(* CODESYS project outputs.project

Project tree, tasks and I/O mapping:
  Device : CODESYS Control Win V3 x64, 3S - Smart Software Solutions GmbH, version 3.5.11.0
    application Application
      libraries: Standard, * (System); VisuDialogs, * (System); Util, * (System)
      task MainTask (cyclic, interval t#10ms, priority 1) calls Plant, Controller
      program Plant [ST]
      global variables GVL
      program Controller [ST]
      visualisation Visualization
      image pool ImagePool
  text list GlobalTextList
  5ce3da45-db07-42e7-a21c-a00fff4ed8f6|C:\Users\mihas\Documents\NSU2026\AM\images\input\beer.png
  5ce3da45-db07-42e7-a21c-a00fff4ed8f6|C:\Users\mihas\Documents\NSU2026\AM\images\input\cigaretes after vki .png
  5ce3da45-db07-42e7-a21c-a00fff4ed8f6|C:\Users\mihas\Documents\NSU2026\AM\images\input\greencard.png
  5ce3da45-db07-42e7-a21c-a00fff4ed8f6|C:\Users\mihas\Documents\NSU2026\AM\images\input\jaguar.png
  5ce3da45-db07-42e7-a21c-a00fff4ed8f6|C:\Users\mihas\Documents\NSU2026\AM\images\input\monster.png
  5ce3da45-db07-42e7-a21c-a00fff4ed8f6|C:\Users\mihas\Documents\NSU2026\AM\images\input\pistol.png
  5ce3da45-db07-42e7-a21c-a00fff4ed8f6|C:\Users\mihas\Documents\NSU2026\AM\images\input\voenbilet.png
*)

// Device/Application/GVL
VAR_GLOBAL
	// Sensors:
	onfloor0:BOOL;		// Elevator at floor 0
	onfloor1:BOOL;		// Elevator at floor 1
	onfloor2:BOOL;		// Elevator at floor 2
	door0closed:BOOL;	// Doors at floor 0 are closed
	door1closed:BOOL;	// Doors at floor 1 are closed
	door2closed:BOOL;	// Doors at floor 2 are closed
	button0:BOOL;		// Call button at floor 0
	button1:BOOL;		// Call button at floor 1
	button2:BOOL;		// Call button at floor 2
	call0:BOOL;			// Request floor 0 from inside the cabin 
	call1:BOOL;			// Request floor 1 from inside the cabin
	call2:BOOL;			// Request floor 2 from inside the cabin
	
	// Actuators:
	up:BOOL;			// Control the elevator to go up
	down:BOOL;			// Control the elevator to go down
	open0:BOOL;			// Open the doors at floor 0
	open1:BOOL;			// Open the doors at floor 1
	open2:BOOL;			// Open the doors at floor 2
	
	call0_LED : BOOL;
	call1_LED : BOOL;
	call2_LED : BOOL;
	
	button0_LED : BOOL;
	button1_LED : BOOL;
	button2_LED : BOOL;
	
	floor0_LED : BOOL;
	floor1_LED : BOOL;
	floor2_LED : BOOL;
	
	cur : INT;
END_VAR

// Device/Application/Plant
PROGRAM Plant

VAR
	cur : BOOL;
	dx : DINT;
	start_time_ms : DINT := TIME_TO_DINT(TIME());
	start_time_text : DINT := TIME_TO_DINT(TIME());
	start_time_angle : DINT := TIME_TO_DINT(TIME());
	angle : DINT := 0;

	sets: STRING := 'TIP TERMINAL';

	i : DINT := 0;
	
	text_welcome_message : WSTRING(250) := "Приветствуем тебя в Пивном Аппарате!!!$nВыбери товар, брат)";
	text_out_of_stock : WSTRING(250) := "В аппарате кончился выбранный товар, брат.$nЗаходи завтра, брат.";
	text_in_stock : WSTRING(250) := "Брат, товар, который ты хочешь есть в наличии.$nЩа оплатить только надо будет, брат.";
	text_insert_payment : WSTRING(250) := "Плати бабки за товар, брат.";
	text_not_enough_money : WSTRING(250) := "Добрось монеток, брат.$nСредств недостаточно.";
	text_stuff_not_dropped : WSTRING(250) := "Пружина не сработала, брат, либо возникла другая проблема.$nПозвони в поддержку, брат. Там всегда ждут твоего звонка";
	text_mission_completed : WSTRING(250) := "Братишка, у тебя получилось.$nНаслаждайся тяжелым люксом, брат!!!";
	
	text_arr : ARRAY[0..6] OF WSTRING(250) := [text_welcome_message, text_out_of_stock, text_in_stock, text_insert_payment, text_not_enough_money, text_stuff_not_dropped, text_mission_completed];
	
	text_display : WSTRING(1024) := text_welcome_message;
	
	Springs : ARRAY [0..4] OF BOOL := [FALSE, FALSE, FALSE, FALSE, FALSE];

END_VAR

dx := (TIME_TO_DINT(TIME()) - start_time_ms) / 1000;
IF ((TIME_TO_DINT(TIME())) - start_time_text) MOD 2000 > 1000 THEN 
	start_time_text := TIME_TO_DINT(TIME());
	IF i = 6 THEN
		i := 0;
	ELSE
		i := i + 1;	
	END_IF
	
	
END_IF

// Поворот пружины

IF ((TIME_TO_DINT(TIME())) - start_time_angle) MOD 2000 > (1000 / 25) THEN 
	start_time_angle := TIME_TO_DINT(TIME());
	angle := (angle + 360 / 25) MOD 360;
END_IF


text_display := text_arr[i];

END_PROGRAM

// Device/Application/Controller
PROGRAM Controller

VAR CONSTANT
	_STOP : INT := 254;
	_ERROR : INT := 255;
END_VAR

VAR
	target : INT;
END_VAR

END_PROGRAM

// Device/Application/Visualization
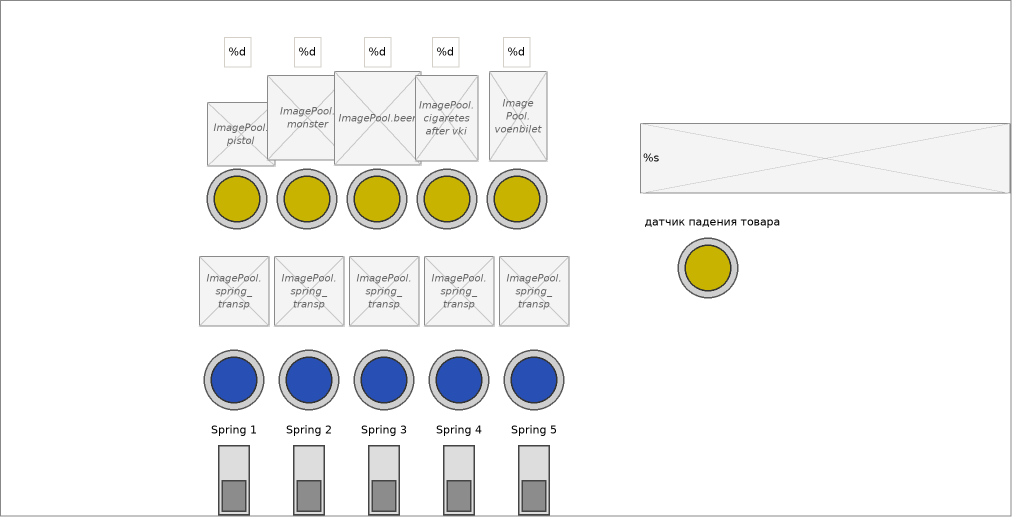
VISUALIZATION Visualization  // 1012x517
    Polygon (363,76) (364,77)
    Lamp1 (199,345 70x70), variable: Plant.Springs[0], style: Lamp-Lamp1-Blue
    Lamp1 (274,345 70x70), variable: Plant.Springs[1], style: Lamp-Lamp1-Blue
    Lamp1 (349,345 70x70), variable: Plant.Springs[2], style: Lamp-Lamp1-Blue
    Lamp1 (424,345 70x70), variable: Plant.Springs[3], style: Lamp-Lamp1-Blue
    Lamp1 (499,345 70x70), variable: Plant.Springs[4], style: Lamp-Lamp1-Blue
    DipSwitch (424,445 70x70), variable: Plant.Springs[3], behaviour: TOGGLE, style: Switch-DipSwitch-Gray
    Image (640,123 370x70), "%s", text variable: Plant.text_display, image: VisuDialogs.ImagePoolDialogs.Title
    Label (199,415 70x30), "Spring 1"
    Label (499,415 70x30), "Spring 5"
    Label (274,415 70x30), "Spring 2"
    Label (349,415 70x30), "Spring 3"
    Label (424,415 70x30), "Spring 4"
    DipSwitch (499,445 70x70), variable: Plant.Springs[4], behaviour: TOGGLE, style: Switch-DipSwitch-Gray
    DipSwitch (349,445 70x70), variable: Plant.Springs[2], behaviour: TOGGLE, style: Switch-DipSwitch-Gray
    DipSwitch (274,445 70x70), variable: Plant.Springs[1], behaviour: TOGGLE, style: Switch-DipSwitch-Gray
    DipSwitch (199,445 70x70), variable: Plant.Springs[0], behaviour: TOGGLE, style: Switch-DipSwitch-Gray
    Image (199,256 70x70), image: ImagePool.spring_transp
    Image (274,256 70x70), image: ImagePool.spring_transp
    Image (349,256 70x70), image: ImagePool.spring_transp
    Image (424,256 70x70), image: ImagePool.spring_transp
    Image (499,256 70x70), image: ImagePool.spring_transp
    Lamp1 (673,233 70x70), variable: Plant.Drop_control, style: Lamp-Lamp1-Yellow
    Label (641,195 143x54), "датчик падения товара"
    Lamp1 (202,164 70x70), variable: Plant.Obj[1], style: Lamp-Lamp1-Yellow
    Lamp1 (272,164 70x70), variable: Plant.Obj[2], style: Lamp-Lamp1-Yellow
    Lamp1 (342,164 70x70), variable: Plant.Obj[3], style: Lamp-Lamp1-Yellow
    Lamp1 (412,164 70x70), variable: Plant.Obj[4], style: Lamp-Lamp1-Yellow
    Lamp1 (482,164 70x70), variable: Plant.Obj[5], style: Lamp-Lamp1-Yellow
    Image (207,102 68x64), angle 35, image: ImagePool.pistol
    Image (267,75 81x85), angle 2, image: ImagePool.monster
    Image (334,71 87x94), image: ImagePool.beer
    Image (489,71 58x90), image: ImagePool.voenbilet
    Textfield (224,37 27x30), "%d", text variable: Plant.tovar[1]
    Image (415,75 63x86), image: ImagePool.cigaretes after vki
    Textfield (294,37 27x30), "%d", text variable: Plant.tovar[2]
    Textfield (364,37 27x30), "%d", text variable: Plant.tovar[3]
    Textfield (432,37 27x30), "%d", text variable: Plant.tovar[4]
    Textfield (503,37 27x30), "%d", text variable: Plant.tovar[5]
END_VISUALIZATION
